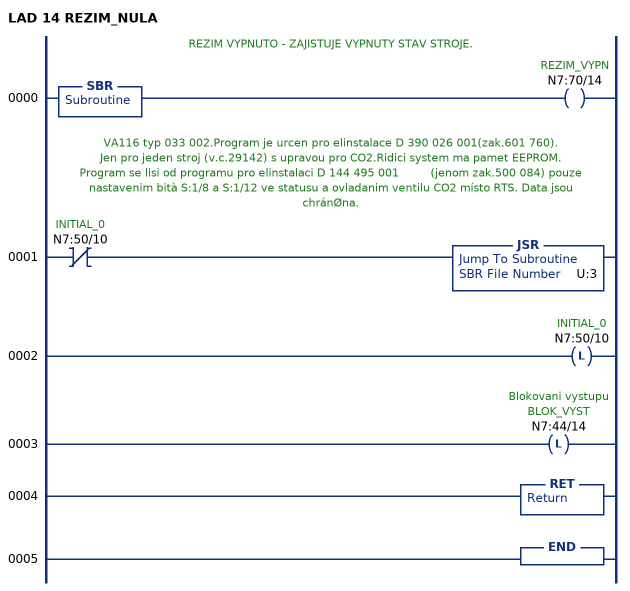
% Rung: 0 %
% REZIM VYPNUTO - ZAJISTUJE VYPNUTY STAV STROJE. %
SOR SBR OTE N7:70/14 EOR
%   N7:70/14  REZIM_VYPN %
% Rung: 1 %
% VA116 typ 033 002.Program je urcen pro elinstalace D 390 026 001(zak.601 760).
% Jen pro jeden stroj (v.c.29142) s upravou pro CO2.Ridici system ma pamet EEPROM. Program se lisi od programu pro elinstalaci D 144 495 001         (jenom zak.500 084) pouze nastavenim bità S:1/8 a S:1/12 ve statusu a ovladanim ventilu CO2 místo RTS. Data jsou chránØna. %
SOR XIO N7:50/10 JSR U:3 EOR
%   N7:50/10  INITIAL_0 %
%   JSR U:3  "Iniciali- zace po zapnuti ridiciho systemu" %
% Rung: 2 %
SOR OTL N7:50/10 EOR
%   N7:50/10  INITIAL_0 %
% Rung: 3 %
SOR OTL N7:44/14 EOR
%   N7:44/14  BLOK_VYST  "Blokovani vystupu" %
% Rung: 4 %
SOR RET EOR
% Rung: 5 %
SOR END EOR

LADDER 15 "STARTSTOP"
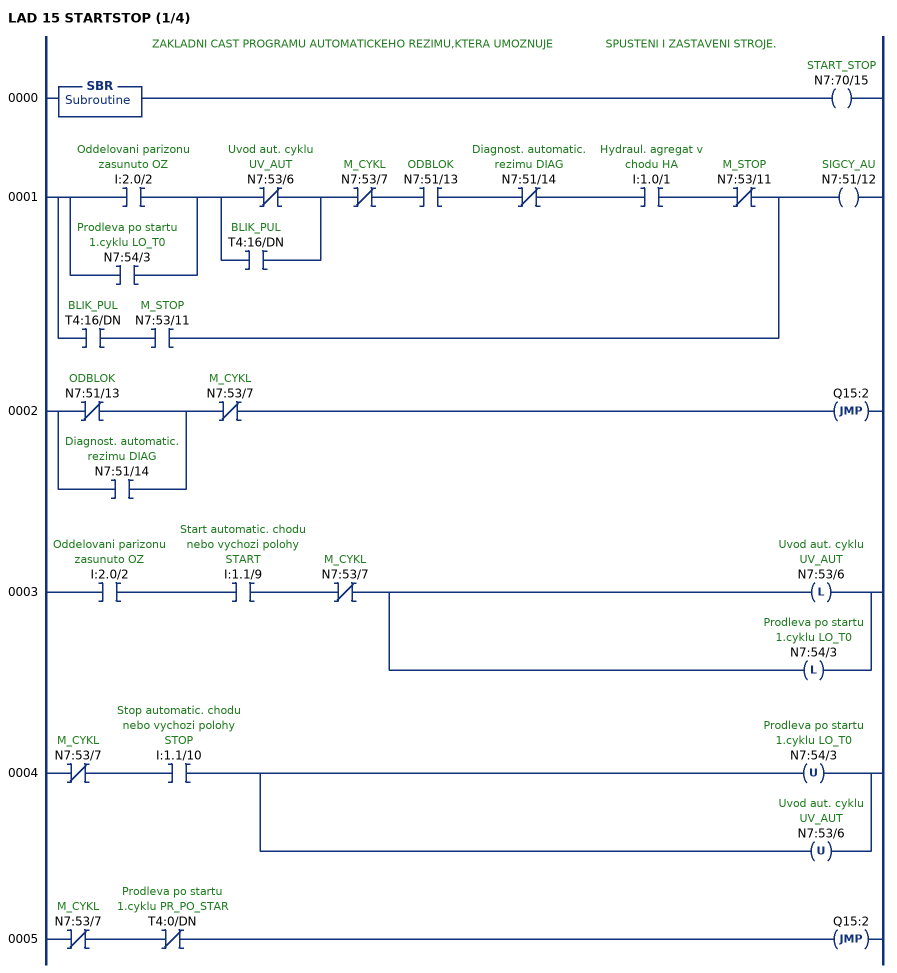
% Rung: 0 %
% ZAKLADNI CAST PROGRAMU AUTOMATICKEHO REZIMU,KTERA UMOZNUJE               SPUSTENI I ZASTAVENI STROJE. %
SOR SBR OTE N7:70/15 EOR
%   N7:70/15  START_STOP %
% Rung: 1 %
SOR BST BST XIC I:2.0/2 NXB XIC N7:54/3 BND BST XIO N7:53/6 NXB XIC T4:16/DN BND XIO N7:53/7 XIC N7:51/13 XIO N7:51/14 XIC I:1.0/1 XIO N7:53/11 NXB XIC T4:16/DN XIC N7:53/11 BND OTE N7:51/12 EOR
%   I:2.0/2  OZ  "Oddelovani parizonu zasunuto" %
%   N7:54/3  LO_T0  "Prodleva po startu 1.cyklu" %
%   N7:53/6  UV_AUT  "Uvod aut. cyklu" %
%   T4:16/DN  BLIK_PUL %
%   N7:53/7  M_CYKL %
%   N7:51/13  ODBLOK %
%   N7:51/14  DIAG  "Diagnost. automatic. rezimu" %
%   I:1.0/1  HA  "Hydraul. agregat v chodu" %
%   N7:53/11  M_STOP %
%   N7:51/12  SIGCY_AU %
% Rung: 2 %
SOR BST XIO N7:51/13 NXB XIC N7:51/14 BND XIO N7:53/7 JMP Q15:2 EOR
%   N7:51/13  ODBLOK %
%   N7:51/14  DIAG  "Diagnost. automatic. rezimu" %
%   N7:53/7  M_CYKL %
% Rung: 3 %
SOR XIC I:2.0/2 XIC I:1.1/9 XIO N7:53/7 BST OTL N7:53/6 NXB OTL N7:54/3 BND EOR
%   I:2.0/2  OZ  "Oddelovani parizonu zasunuto" %
%   I:1.1/9  START  "Start automatic. chodu nebo vychozi polohy" %
%   N7:53/7  M_CYKL %
%   N7:53/6  UV_AUT  "Uvod aut. cyklu" %
%   N7:54/3  LO_T0  "Prodleva po startu 1.cyklu" %
% Rung: 4 %
SOR XIO N7:53/7 XIC I:1.1/10 BST OTU N7:54/3 NXB OTU N7:53/6 BND EOR
%   N7:53/7  M_CYKL %
%   I:1.1/10  STOP  "Stop automatic. chodu nebo vychozi polohy" %
%   N7:54/3  LO_T0  "Prodleva po startu 1.cyklu" %
%   N7:53/6  UV_AUT  "Uvod aut. cyklu" %
% Rung: 5 %
SOR XIO N7:53/7 XIO T4:0/DN JMP Q15:2 EOR
%   N7:53/7  M_CYKL %
%   T4:0/DN  PR_PO_STAR  "Prodleva po startu 1.cyklu" %

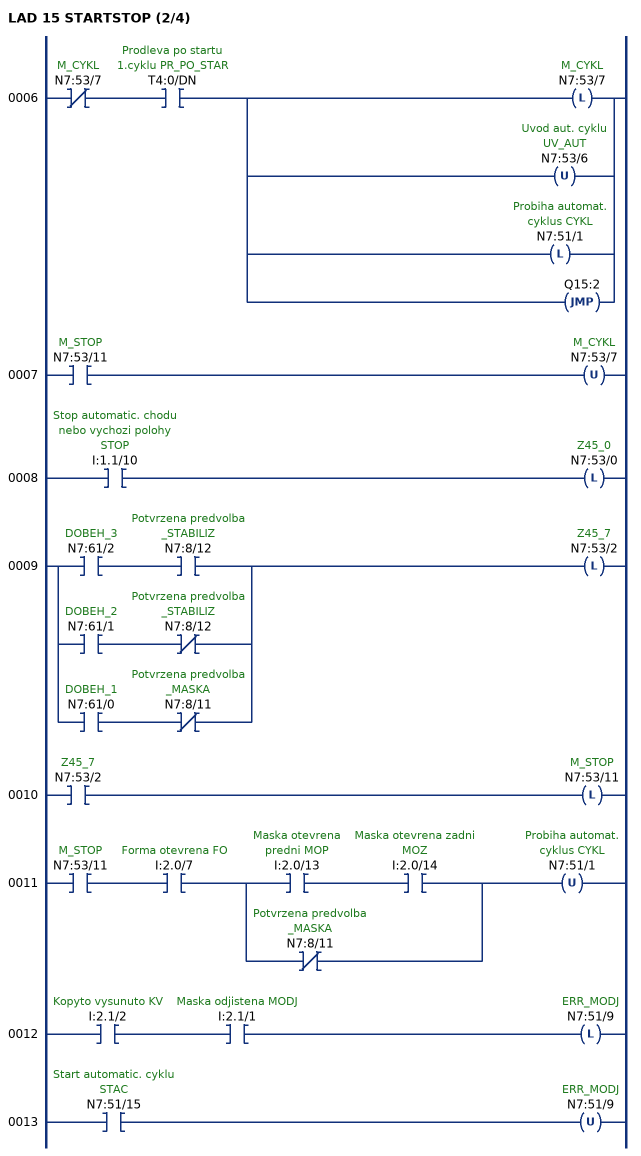
% Rung: 6 %
SOR XIO N7:53/7 XIC T4:0/DN BST OTL N7:53/7 NXB OTU N7:53/6 NXB OTL N7:51/1 NXB JMP Q15:2 BND EOR
%   N7:53/7  M_CYKL %
%   T4:0/DN  PR_PO_STAR  "Prodleva po startu 1.cyklu" %
%   N7:53/6  UV_AUT  "Uvod aut. cyklu" %
%   N7:51/1  CYKL  "Probiha automat. cyklus" %
% Rung: 7 %
SOR XIC N7:53/11 OTU N7:53/7 EOR
%   N7:53/11  M_STOP %
%   N7:53/7  M_CYKL %
% Rung: 8 %
SOR XIC I:1.1/10 OTL N7:53/0 EOR
%   I:1.1/10  STOP  "Stop automatic. chodu nebo vychozi polohy" %
%   N7:53/0  Z45_0 %
% Rung: 9 %
SOR BST XIC N7:61/2 XIC N7:8/12 NXB XIC N7:61/1 XIO N7:8/12 NXB XIC N7:61/0 XIO N7:8/11 BND OTL N7:53/2 EOR
%   N7:61/2  DOBEH_3 %
%   N7:8/12  _STABILIZ  "Potvrzena predvolba" %
%   N7:61/1  DOBEH_2 %
%   N7:61/0  DOBEH_1 %
%   N7:8/11  _MASKA  "Potvrzena predvolba" %
%   N7:53/2  Z45_7 %
% Rung: 10 %
SOR XIC N7:53/2 OTL N7:53/11 EOR
%   N7:53/2  Z45_7 %
%   N7:53/11  M_STOP %
% Rung: 11 %
SOR XIC N7:53/11 XIC I:2.0/7 BST XIC I:2.0/13 XIC I:2.0/14 NXB XIO N7:8/11 BND OTU N7:51/1 EOR
%   N7:53/11  M_STOP %
%   I:2.0/7  FO  "Forma otevrena" %
%   I:2.0/13  MOP  "Maska otevrena predni" %
%   I:2.0/14  MOZ  "Maska otevrena zadni" %
%   N7:8/11  _MASKA  "Potvrzena predvolba" %
%   N7:51/1  CYKL  "Probiha automat. cyklus" %
% Rung: 12 %
SOR XIC I:2.1/2 XIC I:2.1/1 OTL N7:51/9 EOR
%   I:2.1/2  KV  "Kopyto vysunuto" %
%   I:2.1/1  MODJ  "Maska odjistena" %
%   N7:51/9  ERR_MODJ %
% Rung: 13 %
SOR XIC N7:51/15 OTU N7:51/9 EOR
%   N7:51/15  STAC  "Start automatic. cyklu" %
%   N7:51/9  ERR_MODJ %

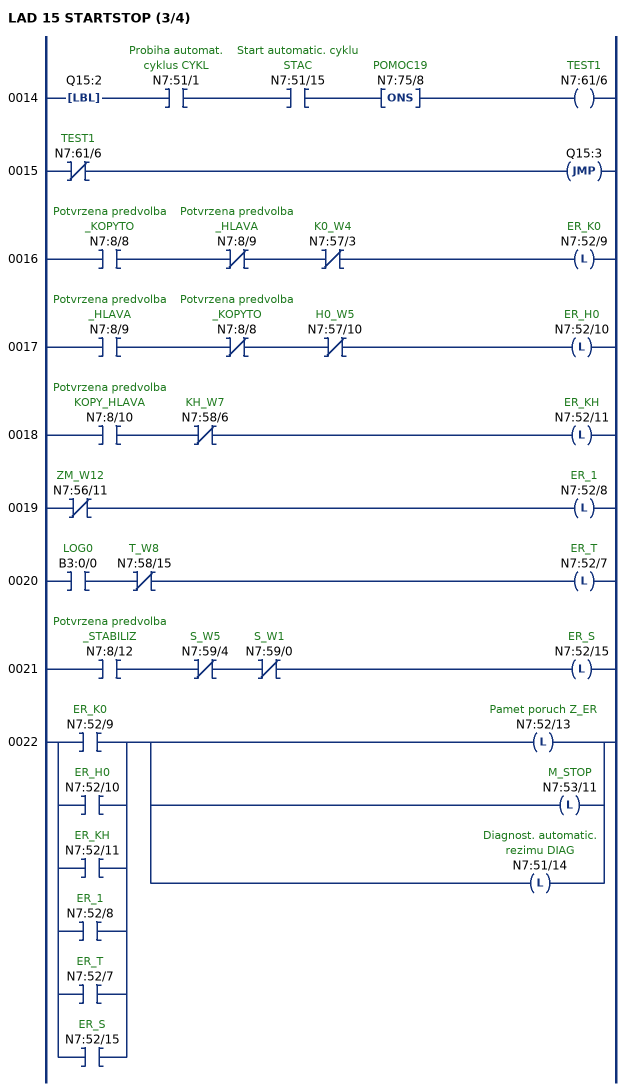
% Rung: 14 %
SOR LBL Q15:2 XIC N7:51/1 XIC N7:51/15 OSR N7:75/8 OTE N7:61/6 EOR
%   N7:51/1  CYKL  "Probiha automat. cyklus" %
%   N7:51/15  STAC  "Start automatic. cyklu" %
%   N7:75/8  POMOC19 %
%   N7:61/6  TEST1 %
% Rung: 15 %
SOR XIO N7:61/6 JMP Q15:3 EOR
%   N7:61/6  TEST1 %
% Rung: 16 %
SOR XIC N7:8/8 XIO N7:8/9 XIO N7:57/3 OTL N7:52/9 EOR
%   N7:8/8  _KOPYTO  "Potvrzena predvolba" %
%   N7:8/9  _HLAVA  "Potvrzena predvolba" %
%   N7:57/3  K0_W4 %
%   N7:52/9  ER_K0 %
% Rung: 17 %
SOR XIC N7:8/9 XIO N7:8/8 XIO N7:57/10 OTL N7:52/10 EOR
%   N7:8/9  _HLAVA  "Potvrzena predvolba" %
%   N7:8/8  _KOPYTO  "Potvrzena predvolba" %
%   N7:57/10  H0_W5 %
%   N7:52/10  ER_H0 %
% Rung: 18 %
SOR XIC N7:8/10 XIO N7:58/6 OTL N7:52/11 EOR
%   N7:8/10  KOPY_HLAVA  "Potvrzena predvolba" %
%   N7:58/6  KH_W7 %
%   N7:52/11  ER_KH %
% Rung: 19 %
SOR XIO N7:56/11 OTL N7:52/8 EOR
%   N7:56/11  ZM_W12 %
%   N7:52/8  ER_1 %
% Rung: 20 %
SOR XIC B3:0/0 XIO N7:58/15 OTL N7:52/7 EOR
%   B3:0/0  LOG0 %
%   N7:58/15  T_W8 %
%   N7:52/7  ER_T %
% Rung: 21 %
SOR XIC N7:8/12 XIO N7:59/4 XIO N7:59/0 OTL N7:52/15 EOR
%   N7:8/12  _STABILIZ  "Potvrzena predvolba" %
%   N7:59/4  S_W5 %
%   N7:59/0  S_W1 %
%   N7:52/15  ER_S %
% Rung: 22 %
SOR BST XIC N7:52/9 NXB XIC N7:52/10 NXB XIC N7:52/11 NXB XIC N7:52/8 NXB XIC N7:52/7 NXB XIC N7:52/15 BND BST OTL N7:52/13 NXB OTL N7:53/11 NXB OTL N7:51/14 BND EOR
%   N7:52/9  ER_K0 %
%   N7:52/10  ER_H0 %
%   N7:52/11  ER_KH %
%   N7:52/8  ER_1 %
%   N7:52/7  ER_T %
%   N7:52/15  ER_S %
%   N7:52/13  Z_ER  "Pamet poruch" %
%   N7:53/11  M_STOP %
%   N7:51/14  DIAG  "Diagnost. automatic. rezimu" %

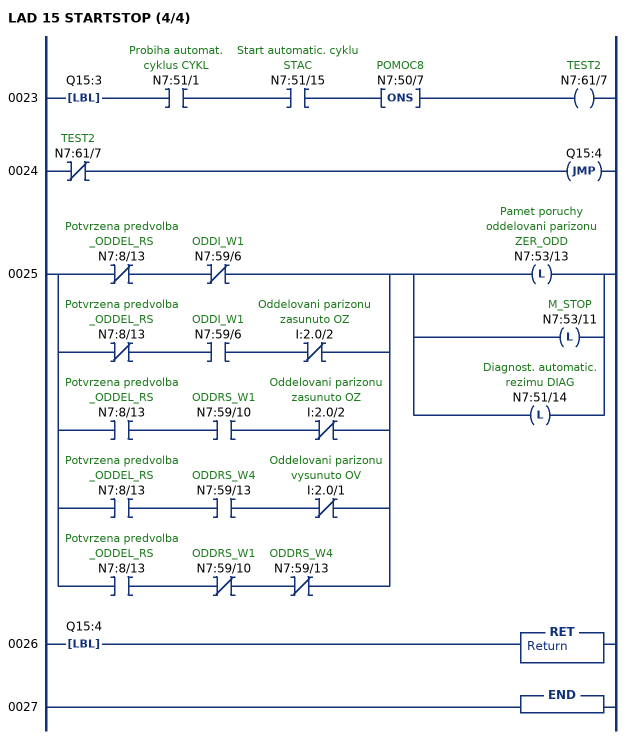
% Rung: 23 %
SOR LBL Q15:3 XIC N7:51/1 XIC N7:51/15 OSR N7:50/7 OTE N7:61/7 EOR
%   N7:51/1  CYKL  "Probiha automat. cyklus" %
%   N7:51/15  STAC  "Start automatic. cyklu" %
%   N7:50/7  POMOC8 %
%   N7:61/7  TEST2 %
% Rung: 24 %
SOR XIO N7:61/7 JMP Q15:4 EOR
%   N7:61/7  TEST2 %
% Rung: 25 %
SOR BST XIO N7:8/13 XIO N7:59/6 NXB XIO N7:8/13 XIC N7:59/6 XIO I:2.0/2 NXB XIC N7:8/13 XIC N7:59/10 XIO I:2.0/2 NXB XIC N7:8/13 XIC N7:59/13 XIO I:2.0/1 NXB XIC N7:8/13 XIO N7:59/10 XIO N7:59/13 BND BST OTL N7:53/13 NXB OTL N7:53/11 NXB OTL N7:51/14 BND EOR
%   N7:8/13  _ODDEL_RS  "Potvrzena predvolba" %
%   N7:59/6  ODDI_W1 %
%   I:2.0/2  OZ  "Oddelovani parizonu zasunuto" %
%   N7:59/10  ODDRS_W1 %
%   N7:59/13  ODDRS_W4 %
%   I:2.0/1  OV  "Oddelovani parizonu vysunuto" %
%   N7:53/13  ZER_ODD  "Pamet poruchy oddelovani parizonu" %
%   N7:53/11  M_STOP %
%   N7:51/14  DIAG  "Diagnost. automatic. rezimu" %
% Rung: 26 %
SOR LBL Q15:4 RET EOR
% Rung: 27 %
SOR END EOR

LADDER 16 "ZAKL_MECH"
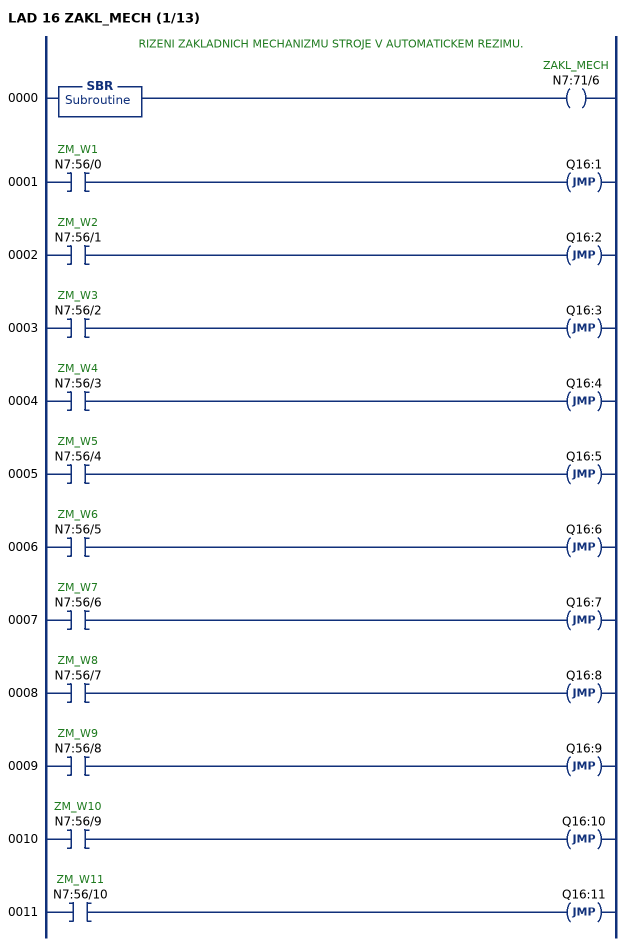
% Rung: 0 %
% RIZENI ZAKLADNICH MECHANIZMU STROJE V AUTOMATICKEM REZIMU. %
SOR SBR OTE N7:71/6 EOR
%   N7:71/6  ZAKL_MECH %
% Rung: 1 %
SOR XIC N7:56/0 JMP Q16:1 EOR
%   N7:56/0  ZM_W1 %
% Rung: 2 %
SOR XIC N7:56/1 JMP Q16:2 EOR
%   N7:56/1  ZM_W2 %
% Rung: 3 %
SOR XIC N7:56/2 JMP Q16:3 EOR
%   N7:56/2  ZM_W3 %
% Rung: 4 %
SOR XIC N7:56/3 JMP Q16:4 EOR
%   N7:56/3  ZM_W4 %
% Rung: 5 %
SOR XIC N7:56/4 JMP Q16:5 EOR
%   N7:56/4  ZM_W5 %
% Rung: 6 %
SOR XIC N7:56/5 JMP Q16:6 EOR
%   N7:56/5  ZM_W6 %
% Rung: 7 %
SOR XIC N7:56/6 JMP Q16:7 EOR
%   N7:56/6  ZM_W7 %
% Rung: 8 %
SOR XIC N7:56/7 JMP Q16:8 EOR
%   N7:56/7  ZM_W8 %
% Rung: 9 %
SOR XIC N7:56/8 JMP Q16:9 EOR
%   N7:56/8  ZM_W9 %
% Rung: 10 %
SOR XIC N7:56/9 JMP Q16:10 EOR
%   N7:56/9  ZM_W10 %
% Rung: 11 %
SOR XIC N7:56/10 JMP Q16:11 EOR
%   N7:56/10  ZM_W11 %

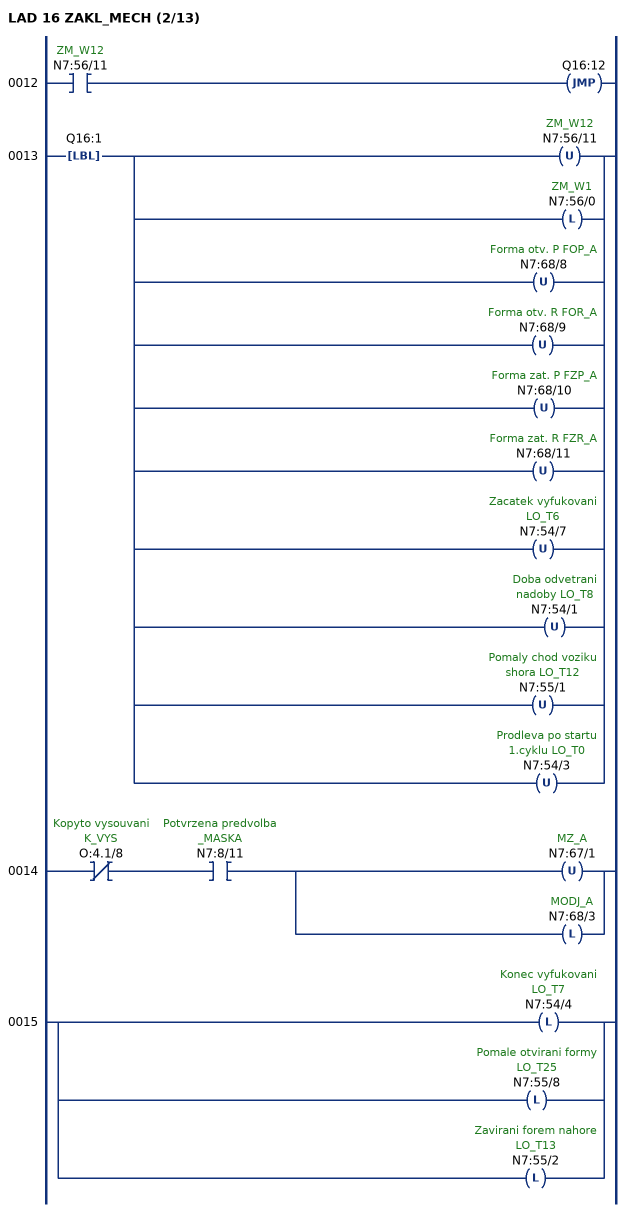
% Rung: 12 %
SOR XIC N7:56/11 JMP Q16:12 EOR
%   N7:56/11  ZM_W12 %
% Rung: 13 %
SOR LBL Q16:1 BST BST OTU N7:56/11 NXB OTL N7:56/0 BND NXB OTU N7:68/8 NXB OTU N7:68/9 NXB OTU N7:68/10 NXB OTU N7:68/11 NXB OTU N7:54/7 NXB OTU N7:54/1 NXB OTU N7:55/1 NXB OTU N7:54/3 BND EOR
%   N7:56/11  ZM_W12 %
%   N7:56/0  ZM_W1 %
%   N7:68/8  FOP_A  "Forma otv. P" %
%   N7:68/9  FOR_A  "Forma otv. R" %
%   N7:68/10  FZP_A  "Forma zat. P" %
%   N7:68/11  FZR_A  "Forma zat. R" %
%   N7:54/7  LO_T6  "Zacatek vyfukovani" %
%   N7:54/1  LO_T8  "Doba odvetrani nadoby" %
%   N7:55/1  LO_T12  "Pomaly chod voziku shora" %
%   N7:54/3  LO_T0  "Prodleva po startu 1.cyklu" %
% Rung: 14 %
SOR XIO O:4.1/8 XIC N7:8/11 BST OTU N7:67/1 NXB OTL N7:68/3 BND EOR
%   O:4.1/8  K_VYS  "Kopyto vysouvani" %
%   N7:8/11  _MASKA  "Potvrzena predvolba" %
%   N7:67/1  MZ_A %
%   N7:68/3  MODJ_A %
% Rung: 15 %
SOR BST OTL N7:54/4 NXB OTL N7:55/8 NXB OTL N7:55/2 BND EOR
%   N7:54/4  LO_T7  "Konec vyfukovani" %
%   N7:55/8  LO_T25  "Pomale otvirani formy" %
%   N7:55/2  LO_T13  "Zavirani forem nahore" %

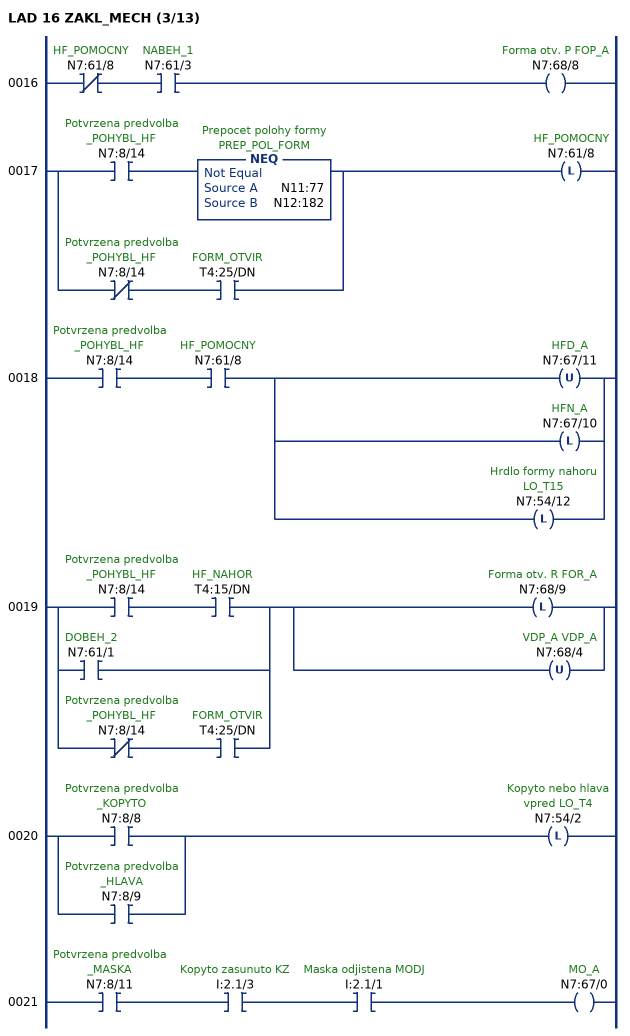
% Rung: 16 %
SOR XIO N7:61/8 XIC N7:61/3 OTE N7:68/8 EOR
%   N7:61/8  HF_POMOCNY %
%   N7:61/3  NABEH_1 %
%   N7:68/8  FOP_A  "Forma otv. P" %
% Rung: 17 %
SOR BST XIC N7:8/14 NEQ N11:77 N12:182 NXB XIO N7:8/14 XIC T4:25/DN BND OTL N7:61/8 EOR
%   N7:8/14  _POHYBL_HF  "Potvrzena predvolba" %
%   N11:77  PREP_POL_FORM  "Prepocet polohy formy" %
%   T4:25/DN  FORM_OTVIR %
%   N7:61/8  HF_POMOCNY %
% Rung: 18 %
SOR XIC N7:8/14 XIC N7:61/8 BST OTU N7:67/11 NXB OTL N7:67/10 NXB OTL N7:54/12 BND EOR
%   N7:8/14  _POHYBL_HF  "Potvrzena predvolba" %
%   N7:61/8  HF_POMOCNY %
%   N7:67/11  HFD_A %
%   N7:67/10  HFN_A %
%   N7:54/12  LO_T15  "Hrdlo formy nahoru" %
% Rung: 19 %
SOR BST XIC N7:8/14 XIC T4:15/DN NXB XIC N7:61/1 NXB XIO N7:8/14 XIC T4:25/DN BND BST OTL N7:68/9 NXB OTU N7:68/4 BND EOR
%   N7:8/14  _POHYBL_HF  "Potvrzena predvolba" %
%   T4:15/DN  HF_NAHOR %
%   N7:61/1  DOBEH_2 %
%   T4:25/DN  FORM_OTVIR %
%   N7:68/9  FOR_A  "Forma otv. R" %
%   N7:68/4  VDP_A  "VDP_A" %
% Rung: 20 %
SOR BST XIC N7:8/8 NXB XIC N7:8/9 BND OTL N7:54/2 EOR
%   N7:8/8  _KOPYTO  "Potvrzena predvolba" %
%   N7:8/9  _HLAVA  "Potvrzena predvolba" %
%   N7:54/2  LO_T4  "Kopyto nebo hlava vpred" %
% Rung: 21 %
SOR XIC N7:8/11 XIC I:2.1/3 XIC I:2.1/1 OTE N7:67/0 EOR
%   N7:8/11  _MASKA  "Potvrzena predvolba" %
%   I:2.1/3  KZ  "Kopyto zasunuto" %
%   I:2.1/1  MODJ  "Maska odjistena" %
%   N7:67/0  MO_A %

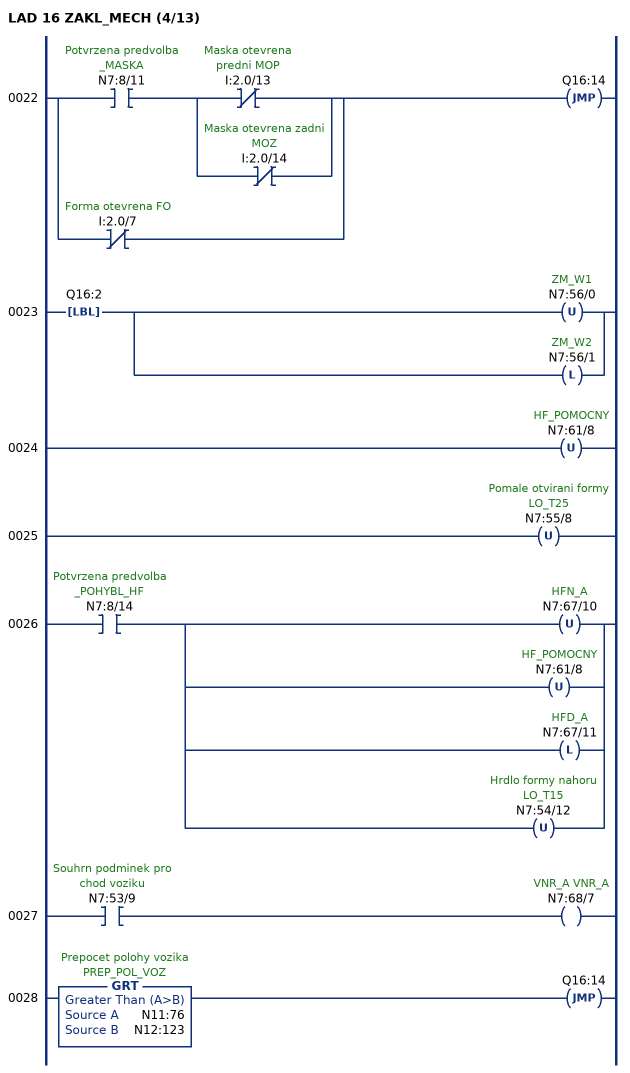
% Rung: 22 %
SOR BST XIC N7:8/11 BST XIO I:2.0/13 NXB XIO I:2.0/14 BND NXB XIO I:2.0/7 BND JMP Q16:14 EOR
%   N7:8/11  _MASKA  "Potvrzena predvolba" %
%   I:2.0/13  MOP  "Maska otevrena predni" %
%   I:2.0/14  MOZ  "Maska otevrena zadni" %
%   I:2.0/7  FO  "Forma otevrena" %
% Rung: 23 %
SOR LBL Q16:2 BST OTU N7:56/0 NXB OTL N7:56/1 BND EOR
%   N7:56/0  ZM_W1 %
%   N7:56/1  ZM_W2 %
% Rung: 24 %
SOR OTU N7:61/8 EOR
%   N7:61/8  HF_POMOCNY %
% Rung: 25 %
SOR OTU N7:55/8 EOR
%   N7:55/8  LO_T25  "Pomale otvirani formy" %
% Rung: 26 %
SOR XIC N7:8/14 BST OTU N7:67/10 NXB OTU N7:61/8 NXB OTL N7:67/11 NXB OTU N7:54/12 BND EOR
%   N7:8/14  _POHYBL_HF  "Potvrzena predvolba" %
%   N7:67/10  HFN_A %
%   N7:61/8  HF_POMOCNY %
%   N7:67/11  HFD_A %
%   N7:54/12  LO_T15  "Hrdlo formy nahoru" %
% Rung: 27 %
SOR XIC N7:53/9 OTE N7:68/7 EOR
%   N7:53/9  "Souhrn podminek pro chod voziku" %
%   N7:68/7  VNR_A  "VNR_A" %
% Rung: 28 %
SOR GRT N11:76 N12:123 JMP Q16:14 EOR
%   N11:76  PREP_POL_VOZ  "Prepocet polohy vozika" %
%   N12:123  N123  "Žiadana poloha vozika c.4 hore" %

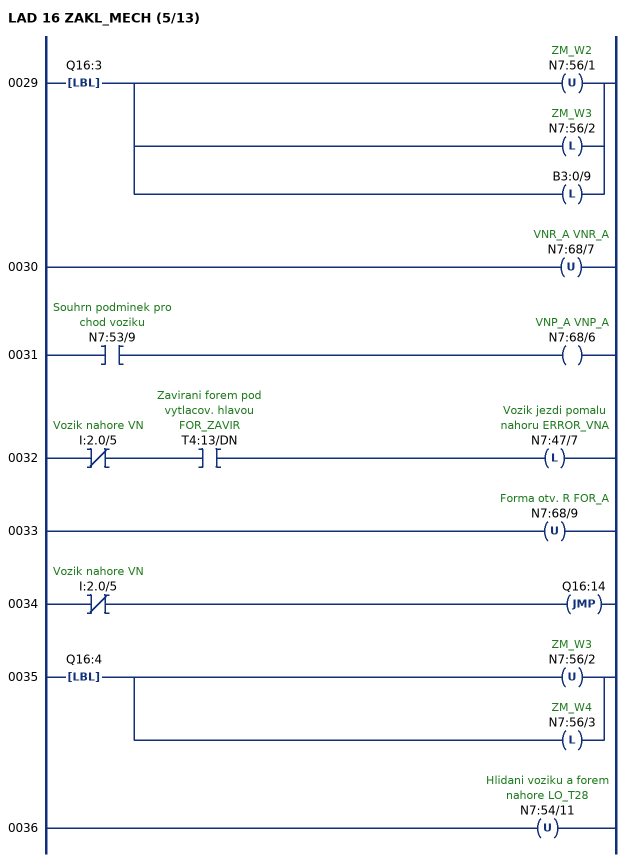
% Rung: 29 %
SOR LBL Q16:3 BST OTU N7:56/1 NXB OTL N7:56/2 NXB OTL B3:0/9 BND EOR
%   N7:56/1  ZM_W2 %
%   N7:56/2  ZM_W3 %
% Rung: 30 %
SOR OTU N7:68/7 EOR
%   N7:68/7  VNR_A  "VNR_A" %
% Rung: 31 %
SOR XIC N7:53/9 OTE N7:68/6 EOR
%   N7:53/9  "Souhrn podminek pro chod voziku" %
%   N7:68/6  VNP_A  "VNP_A" %
% Rung: 32 %
SOR XIO I:2.0/5 XIC T4:13/DN OTL N7:47/7 EOR
%   I:2.0/5  VN  "Vozik nahore" %
%   T4:13/DN  FOR_ZAVIR  "Zavirani forem pod vytlacov. hlavou" %
%   N7:47/7  ERROR_VNA  "Vozik jezdi pomalu nahoru" %
% Rung: 33 %
SOR OTU N7:68/9 EOR
%   N7:68/9  FOR_A  "Forma otv. R" %
% Rung: 34 %
SOR XIO I:2.0/5 JMP Q16:14 EOR
%   I:2.0/5  VN  "Vozik nahore" %
% Rung: 35 %
SOR LBL Q16:4 BST OTU N7:56/2 NXB OTL N7:56/3 BND EOR
%   N7:56/2  ZM_W3 %
%   N7:56/3  ZM_W4 %
% Rung: 36 %
SOR OTU N7:54/11 EOR
%   N7:54/11  LO_T28  "Hlidani voziku a forem nahore" %

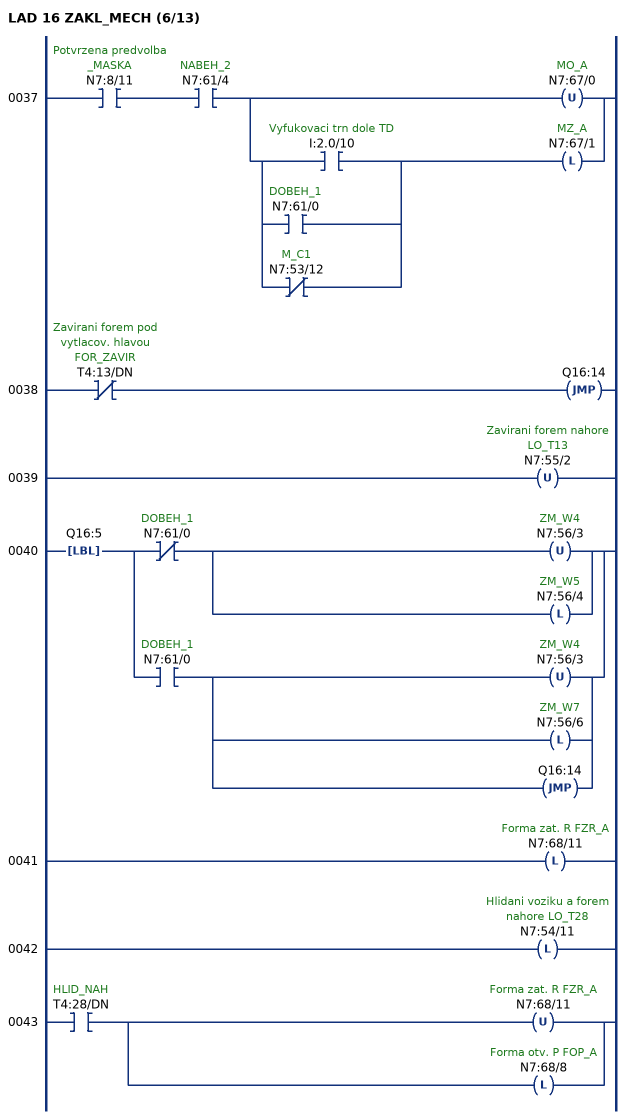
% Rung: 37 %
SOR XIC N7:8/11 XIC N7:61/4 BST OTU N7:67/0 NXB BST XIC I:2.0/10 NXB XIC N7:61/0 NXB XIO N7:53/12 BND OTL N7:67/1 BND EOR
%   N7:8/11  _MASKA  "Potvrzena predvolba" %
%   N7:61/4  NABEH_2 %
%   N7:67/0  MO_A %
%   I:2.0/10  TD  "Vyfukovaci trn dole" %
%   N7:61/0  DOBEH_1 %
%   N7:53/12  M_C1 %
%   N7:67/1  MZ_A %
% Rung: 38 %
SOR XIO T4:13/DN JMP Q16:14 EOR
%   T4:13/DN  FOR_ZAVIR  "Zavirani forem pod vytlacov. hlavou" %
% Rung: 39 %
SOR OTU N7:55/2 EOR
%   N7:55/2  LO_T13  "Zavirani forem nahore" %
% Rung: 40 %
SOR LBL Q16:5 BST XIO N7:61/0 BST OTU N7:56/3 NXB OTL N7:56/4 BND NXB XIC N7:61/0 BST OTU N7:56/3 NXB OTL N7:56/6 NXB JMP Q16:14 BND BND EOR
%   N7:61/0  DOBEH_1 %
%   N7:56/3  ZM_W4 %
%   N7:56/4  ZM_W5 %
%   N7:56/6  ZM_W7 %
% Rung: 41 %
SOR OTL N7:68/11 EOR
%   N7:68/11  FZR_A  "Forma zat. R" %
% Rung: 42 %
SOR OTL N7:54/11 EOR
%   N7:54/11  LO_T28  "Hlidani voziku a forem nahore" %
% Rung: 43 %
SOR XIC T4:28/DN BST OTU N7:68/11 NXB OTL N7:68/8 BND EOR
%   T4:28/DN  HLID_NAH %
%   N7:68/11  FZR_A  "Forma zat. R" %
%   N7:68/8  FOP_A  "Forma otv. P" %

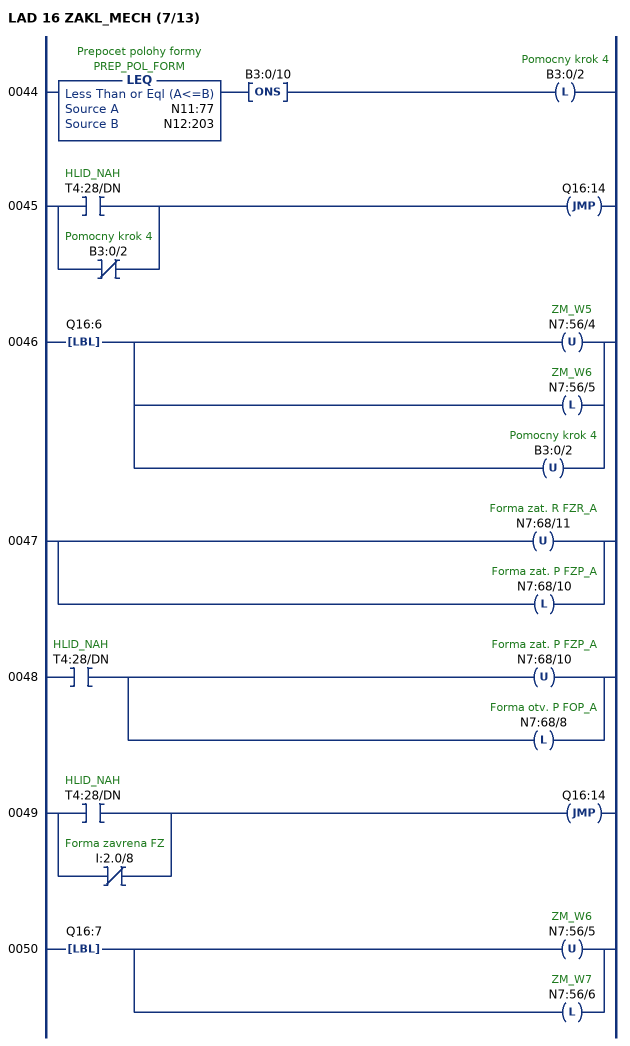
% Rung: 44 %
SOR LEQ N11:77 N12:203 OSR B3:0/10 OTL B3:0/2 EOR
%   N11:77  PREP_POL_FORM  "Prepocet polohy formy" %
%   B3:0/2  "Pomocny krok 4" %
% Rung: 45 %
SOR BST XIC T4:28/DN NXB XIO B3:0/2 BND JMP Q16:14 EOR
%   T4:28/DN  HLID_NAH %
%   B3:0/2  "Pomocny krok 4" %
% Rung: 46 %
SOR LBL Q16:6 BST OTU N7:56/4 NXB OTL N7:56/5 NXB OTU B3:0/2 BND EOR
%   N7:56/4  ZM_W5 %
%   N7:56/5  ZM_W6 %
%   B3:0/2  "Pomocny krok 4" %
% Rung: 47 %
SOR BST OTU N7:68/11 NXB OTL N7:68/10 BND EOR
%   N7:68/11  FZR_A  "Forma zat. R" %
%   N7:68/10  FZP_A  "Forma zat. P" %
% Rung: 48 %
SOR XIC T4:28/DN BST OTU N7:68/10 NXB OTL N7:68/8 BND EOR
%   T4:28/DN  HLID_NAH %
%   N7:68/10  FZP_A  "Forma zat. P" %
%   N7:68/8  FOP_A  "Forma otv. P" %
% Rung: 49 %
SOR BST XIC T4:28/DN NXB XIO I:2.0/8 BND JMP Q16:14 EOR
%   T4:28/DN  HLID_NAH %
%   I:2.0/8  FZ  "Forma zavrena" %
% Rung: 50 %
SOR LBL Q16:7 BST OTU N7:56/5 NXB OTL N7:56/6 BND EOR
%   N7:56/5  ZM_W6 %
%   N7:56/6  ZM_W7 %

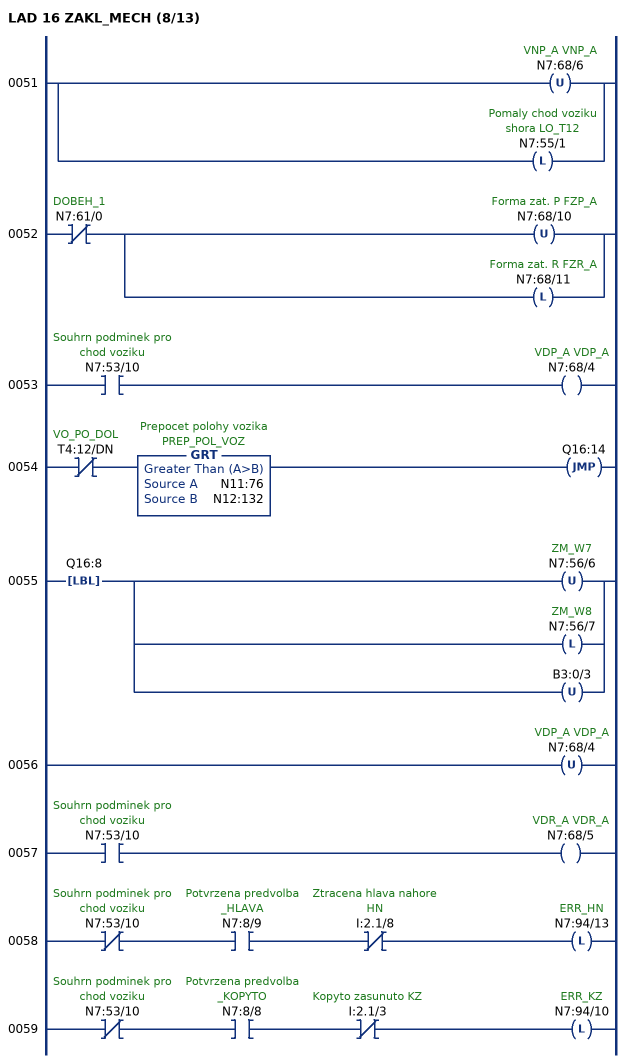
% Rung: 51 %
SOR BST OTU N7:68/6 NXB OTL N7:55/1 BND EOR
%   N7:68/6  VNP_A  "VNP_A" %
%   N7:55/1  LO_T12  "Pomaly chod voziku shora" %
% Rung: 52 %
SOR XIO N7:61/0 BST OTU N7:68/10 NXB OTL N7:68/11 BND EOR
%   N7:61/0  DOBEH_1 %
%   N7:68/10  FZP_A  "Forma zat. P" %
%   N7:68/11  FZR_A  "Forma zat. R" %
% Rung: 53 %
SOR XIC N7:53/10 OTE N7:68/4 EOR
%   N7:53/10  "Souhrn podminek pro chod voziku" %
%   N7:68/4  VDP_A  "VDP_A" %
% Rung: 54 %
SOR XIO T4:12/DN GRT N11:76 N12:132 JMP Q16:14 EOR
%   T4:12/DN  VO_PO_DOL %
%   N11:76  PREP_POL_VOZ  "Prepocet polohy vozika" %
% Rung: 55 %
SOR LBL Q16:8 BST OTU N7:56/6 NXB OTL N7:56/7 NXB OTU B3:0/3 BND EOR
%   N7:56/6  ZM_W7 %
%   N7:56/7  ZM_W8 %
% Rung: 56 %
SOR OTU N7:68/4 EOR
%   N7:68/4  VDP_A  "VDP_A" %
% Rung: 57 %
SOR XIC N7:53/10 OTE N7:68/5 EOR
%   N7:53/10  "Souhrn podminek pro chod voziku" %
%   N7:68/5  VDR_A  "VDR_A" %
% Rung: 58 %
SOR XIO N7:53/10 XIC N7:8/9 XIO I:2.1/8 OTL N7:94/13 EOR
%   N7:53/10  "Souhrn podminek pro chod voziku" %
%   N7:8/9  _HLAVA  "Potvrzena predvolba" %
%   I:2.1/8  HN  "Ztracena hlava nahore" %
%   N7:94/13  ERR_HN %
% Rung: 59 %
SOR XIO N7:53/10 XIC N7:8/8 XIO I:2.1/3 OTL N7:94/10 EOR
%   N7:53/10  "Souhrn podminek pro chod voziku" %
%   N7:8/8  _KOPYTO  "Potvrzena predvolba" %
%   I:2.1/3  KZ  "Kopyto zasunuto" %
%   N7:94/10  ERR_KZ %

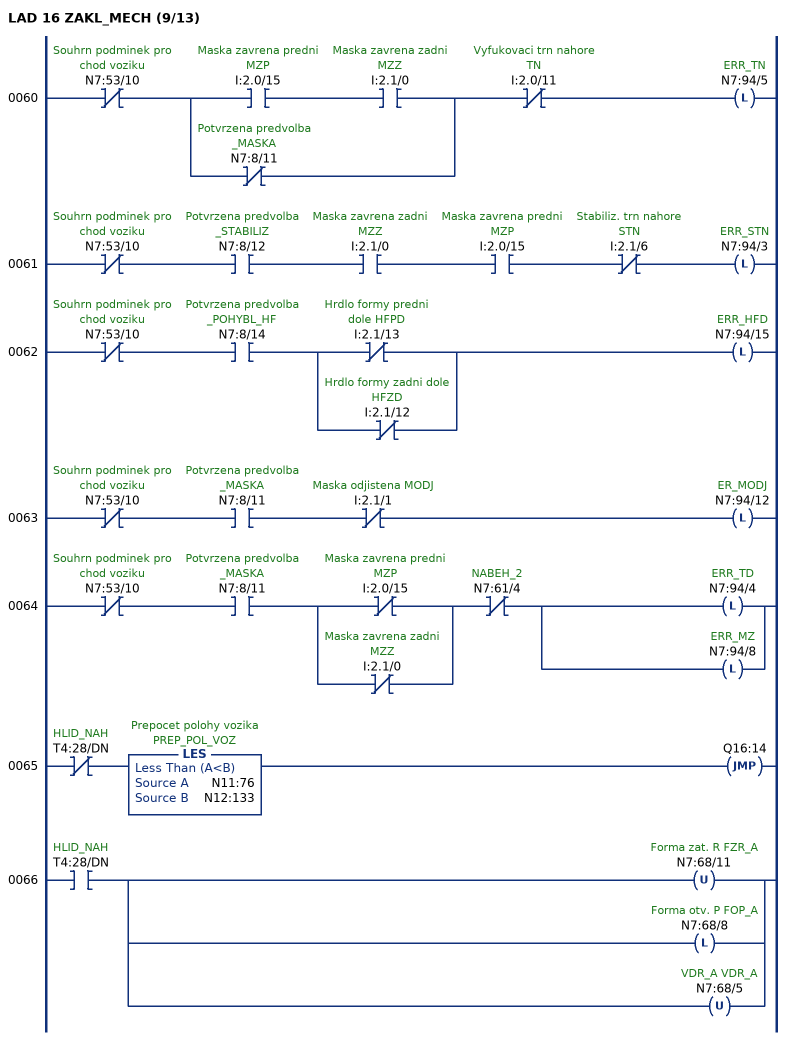
% Rung: 60 %
SOR XIO N7:53/10 BST XIC I:2.0/15 XIC I:2.1/0 NXB XIO N7:8/11 BND XIO I:2.0/11 OTL N7:94/5 EOR
%   N7:53/10  "Souhrn podminek pro chod voziku" %
%   I:2.0/15  MZP  "Maska zavrena predni" %
%   I:2.1/0  MZZ  "Maska zavrena zadni" %
%   N7:8/11  _MASKA  "Potvrzena predvolba" %
%   I:2.0/11  TN  "Vyfukovaci trn nahore" %
%   N7:94/5  ERR_TN %
% Rung: 61 %
SOR XIO N7:53/10 XIC N7:8/12 XIC I:2.1/0 XIC I:2.0/15 XIO I:2.1/6 OTL N7:94/3 EOR
%   N7:53/10  "Souhrn podminek pro chod voziku" %
%   N7:8/12  _STABILIZ  "Potvrzena predvolba" %
%   I:2.1/0  MZZ  "Maska zavrena zadni" %
%   I:2.0/15  MZP  "Maska zavrena predni" %
%   I:2.1/6  STN  "Stabiliz. trn nahore" %
%   N7:94/3  ERR_STN %
% Rung: 62 %
SOR XIO N7:53/10 XIC N7:8/14 BST XIO I:2.1/13 NXB XIO I:2.1/12 BND OTL N7:94/15 EOR
%   N7:53/10  "Souhrn podminek pro chod voziku" %
%   N7:8/14  _POHYBL_HF  "Potvrzena predvolba" %
%   I:2.1/13  HFPD  "Hrdlo formy predni dole" %
%   I:2.1/12  HFZD  "Hrdlo formy zadni dole" %
%   N7:94/15  ERR_HFD %
% Rung: 63 %
SOR XIO N7:53/10 XIC N7:8/11 XIO I:2.1/1 OTL N7:94/12 EOR
%   N7:53/10  "Souhrn podminek pro chod voziku" %
%   N7:8/11  _MASKA  "Potvrzena predvolba" %
%   I:2.1/1  MODJ  "Maska odjistena" %
%   N7:94/12  ER_MODJ %
% Rung: 64 %
SOR XIO N7:53/10 XIC N7:8/11 BST XIO I:2.0/15 NXB XIO I:2.1/0 BND XIO N7:61/4 BST OTL N7:94/4 NXB OTL N7:94/8 BND EOR
%   N7:53/10  "Souhrn podminek pro chod voziku" %
%   N7:8/11  _MASKA  "Potvrzena predvolba" %
%   I:2.0/15  MZP  "Maska zavrena predni" %
%   I:2.1/0  MZZ  "Maska zavrena zadni" %
%   N7:61/4  NABEH_2 %
%   N7:94/4  ERR_TD %
%   N7:94/8  ERR_MZ %
% Rung: 65 %
SOR XIO T4:28/DN LES N11:76 N12:133 JMP Q16:14 EOR
%   T4:28/DN  HLID_NAH %
%   N11:76  PREP_POL_VOZ  "Prepocet polohy vozika" %
% Rung: 66 %
SOR XIC T4:28/DN BST OTU N7:68/11 NXB OTL N7:68/8 NXB OTU N7:68/5 BND EOR
%   T4:28/DN  HLID_NAH %
%   N7:68/11  FZR_A  "Forma zat. R" %
%   N7:68/8  FOP_A  "Forma otv. P" %
%   N7:68/5  VDR_A  "VDR_A" %

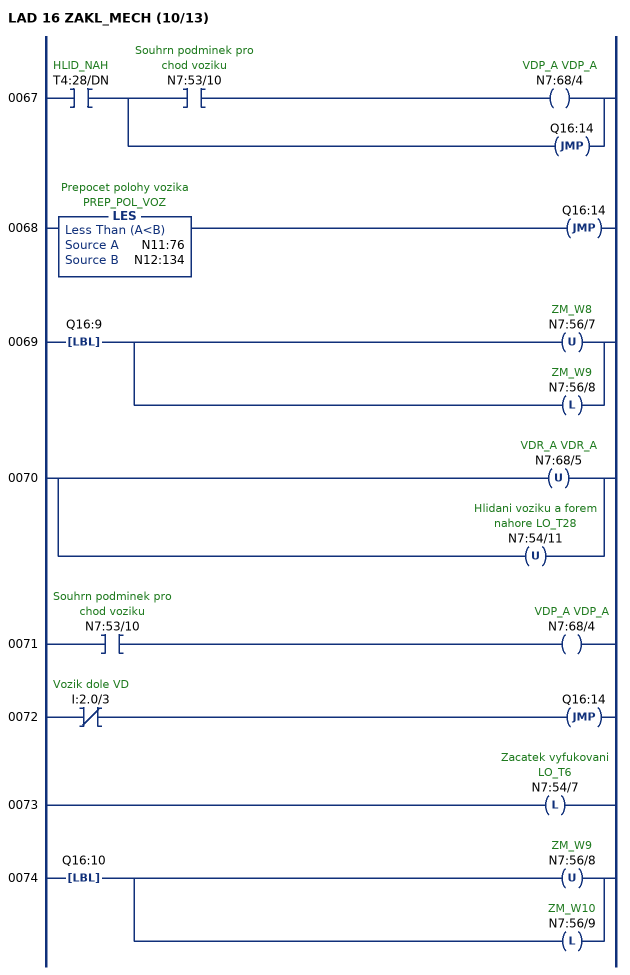
% Rung: 67 %
SOR XIC T4:28/DN BST XIC N7:53/10 OTE N7:68/4 NXB JMP Q16:14 BND EOR
%   T4:28/DN  HLID_NAH %
%   N7:53/10  "Souhrn podminek pro chod voziku" %
%   N7:68/4  VDP_A  "VDP_A" %
% Rung: 68 %
SOR LES N11:76 N12:134 JMP Q16:14 EOR
%   N11:76  PREP_POL_VOZ  "Prepocet polohy vozika" %
% Rung: 69 %
SOR LBL Q16:9 BST OTU N7:56/7 NXB OTL N7:56/8 BND EOR
%   N7:56/7  ZM_W8 %
%   N7:56/8  ZM_W9 %
% Rung: 70 %
SOR BST OTU N7:68/5 NXB OTU N7:54/11 BND EOR
%   N7:68/5  VDR_A  "VDR_A" %
%   N7:54/11  LO_T28  "Hlidani voziku a forem nahore" %
% Rung: 71 %
SOR XIC N7:53/10 OTE N7:68/4 EOR
%   N7:53/10  "Souhrn podminek pro chod voziku" %
%   N7:68/4  VDP_A  "VDP_A" %
% Rung: 72 %
SOR XIO I:2.0/3 JMP Q16:14 EOR
%   I:2.0/3  VD  "Vozik dole" %
% Rung: 73 %
SOR OTL N7:54/7 EOR
%   N7:54/7  LO_T6  "Zacatek vyfukovani" %
% Rung: 74 %
SOR LBL Q16:10 BST OTU N7:56/8 NXB OTL N7:56/9 BND EOR
%   N7:56/8  ZM_W9 %
%   N7:56/9  ZM_W10 %

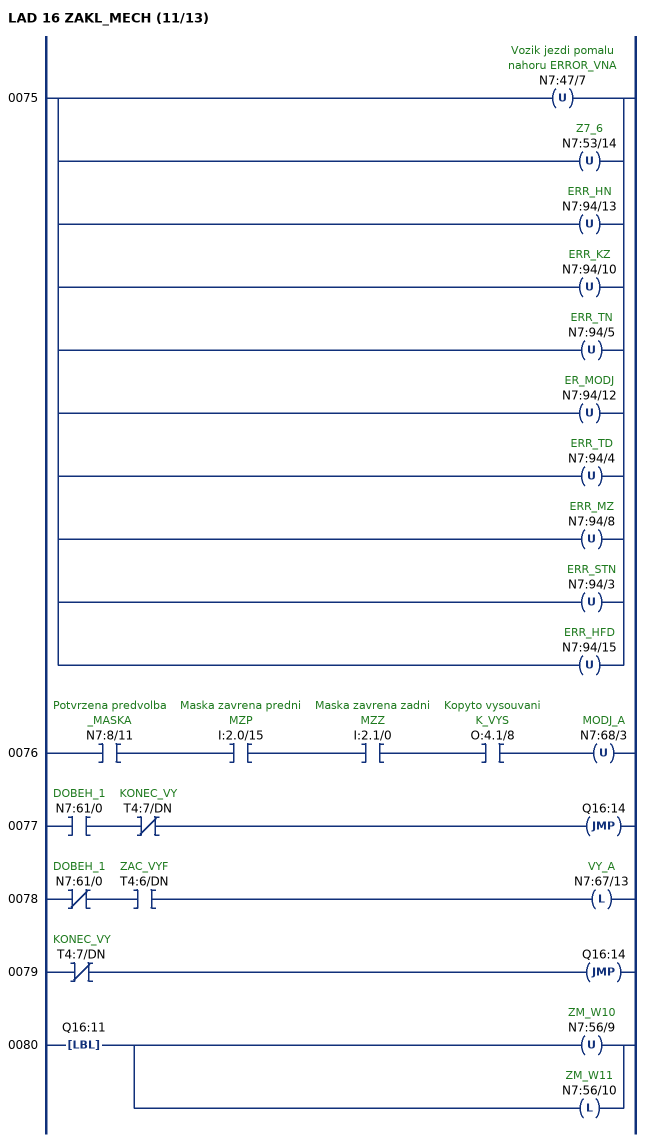
% Rung: 75 %
SOR BST OTU N7:47/7 NXB OTU N7:53/14 NXB OTU N7:94/13 NXB OTU N7:94/10 NXB OTU N7:94/5 NXB OTU N7:94/12 NXB OTU N7:94/4 NXB OTU N7:94/8 NXB OTU N7:94/3 NXB OTU N7:94/15 BND EOR
%   N7:47/7  ERROR_VNA  "Vozik jezdi pomalu nahoru" %
%   N7:53/14  Z7_6 %
%   N7:94/13  ERR_HN %
%   N7:94/10  ERR_KZ %
%   N7:94/5  ERR_TN %
%   N7:94/12  ER_MODJ %
%   N7:94/4  ERR_TD %
%   N7:94/8  ERR_MZ %
%   N7:94/3  ERR_STN %
%   N7:94/15  ERR_HFD %
% Rung: 76 %
SOR XIC N7:8/11 XIC I:2.0/15 XIC I:2.1/0 XIC O:4.1/8 OTU N7:68/3 EOR
%   N7:8/11  _MASKA  "Potvrzena predvolba" %
%   I:2.0/15  MZP  "Maska zavrena predni" %
%   I:2.1/0  MZZ  "Maska zavrena zadni" %
%   O:4.1/8  K_VYS  "Kopyto vysouvani" %
%   N7:68/3  MODJ_A %
% Rung: 77 %
SOR XIC N7:61/0 XIO T4:7/DN JMP Q16:14 EOR
%   N7:61/0  DOBEH_1 %
%   T4:7/DN  KONEC_VY %
% Rung: 78 %
SOR XIO N7:61/0 XIC T4:6/DN OTL N7:67/13 EOR
%   N7:61/0  DOBEH_1 %
%   T4:6/DN  ZAC_VYF %
%   N7:67/13  VY_A %
% Rung: 79 %
SOR XIO T4:7/DN JMP Q16:14 EOR
%   T4:7/DN  KONEC_VY %
% Rung: 80 %
SOR LBL Q16:11 BST OTU N7:56/9 NXB OTL N7:56/10 BND EOR
%   N7:56/9  ZM_W10 %
%   N7:56/10  ZM_W11 %

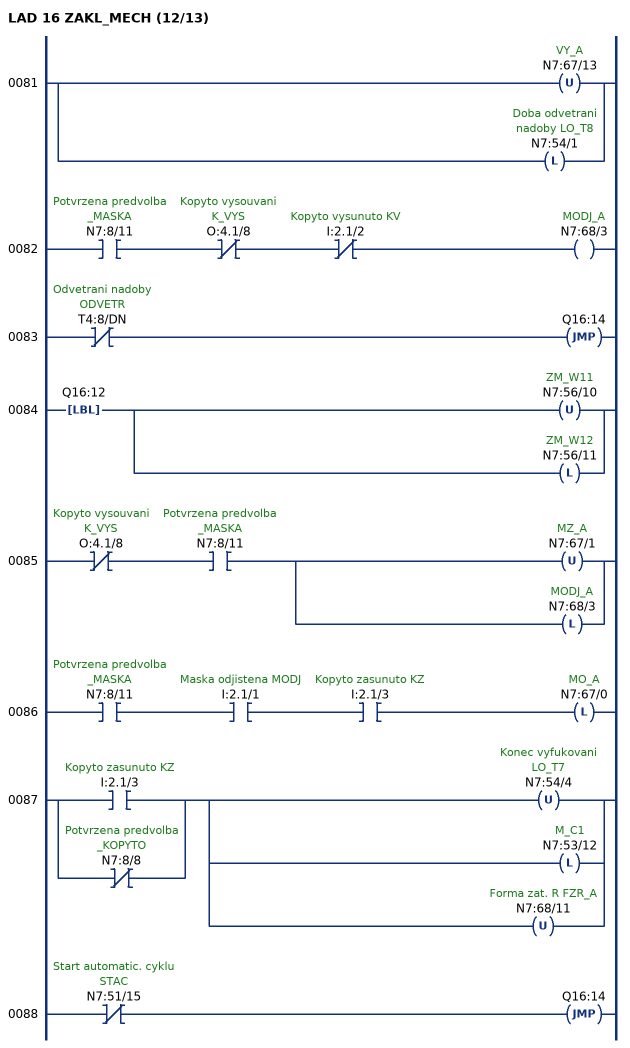
% Rung: 81 %
SOR BST OTU N7:67/13 NXB OTL N7:54/1 BND EOR
%   N7:67/13  VY_A %
%   N7:54/1  LO_T8  "Doba odvetrani nadoby" %
% Rung: 82 %
SOR XIC N7:8/11 XIO O:4.1/8 XIO I:2.1/2 OTE N7:68/3 EOR
%   N7:8/11  _MASKA  "Potvrzena predvolba" %
%   O:4.1/8  K_VYS  "Kopyto vysouvani" %
%   I:2.1/2  KV  "Kopyto vysunuto" %
%   N7:68/3  MODJ_A %
% Rung: 83 %
SOR XIO T4:8/DN JMP Q16:14 EOR
%   T4:8/DN  ODVETR  "Odvetrani nadoby" %
% Rung: 84 %
SOR LBL Q16:12 BST OTU N7:56/10 NXB OTL N7:56/11 BND EOR
%   N7:56/10  ZM_W11 %
%   N7:56/11  ZM_W12 %
% Rung: 85 %
SOR XIO O:4.1/8 XIC N7:8/11 BST OTU N7:67/1 NXB OTL N7:68/3 BND EOR
%   O:4.1/8  K_VYS  "Kopyto vysouvani" %
%   N7:8/11  _MASKA  "Potvrzena predvolba" %
%   N7:67/1  MZ_A %
%   N7:68/3  MODJ_A %
% Rung: 86 %
SOR XIC N7:8/11 XIC I:2.1/1 XIC I:2.1/3 OTL N7:67/0 EOR
%   N7:8/11  _MASKA  "Potvrzena predvolba" %
%   I:2.1/1  MODJ  "Maska odjistena" %
%   I:2.1/3  KZ  "Kopyto zasunuto" %
%   N7:67/0  MO_A %
% Rung: 87 %
SOR BST XIC I:2.1/3 NXB XIO N7:8/8 BND BST OTU N7:54/4 NXB OTL N7:53/12 NXB OTU N7:68/11 BND EOR
%   I:2.1/3  KZ  "Kopyto zasunuto" %
%   N7:8/8  _KOPYTO  "Potvrzena predvolba" %
%   N7:54/4  LO_T7  "Konec vyfukovani" %
%   N7:53/12  M_C1 %
%   N7:68/11  FZR_A  "Forma zat. R" %
% Rung: 88 %
SOR XIO N7:51/15 JMP Q16:14 EOR
%   N7:51/15  STAC  "Start automatic. cyklu" %

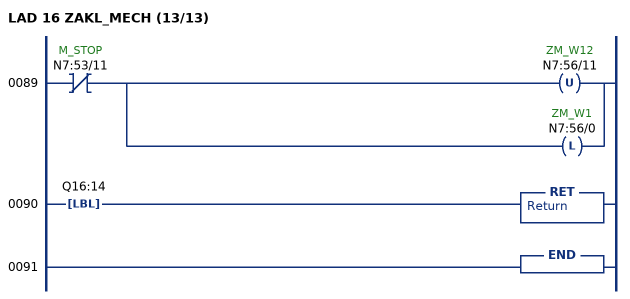
% Rung: 89 %
SOR XIO N7:53/11 BST OTU N7:56/11 NXB OTL N7:56/0 BND EOR
%   N7:53/11  M_STOP %
%   N7:56/11  ZM_W12 %
%   N7:56/0  ZM_W1 %
% Rung: 90 %
SOR LBL Q16:14 RET EOR
% Rung: 91 %
SOR END EOR

LADDER 17 "KOPYTO_SOL"
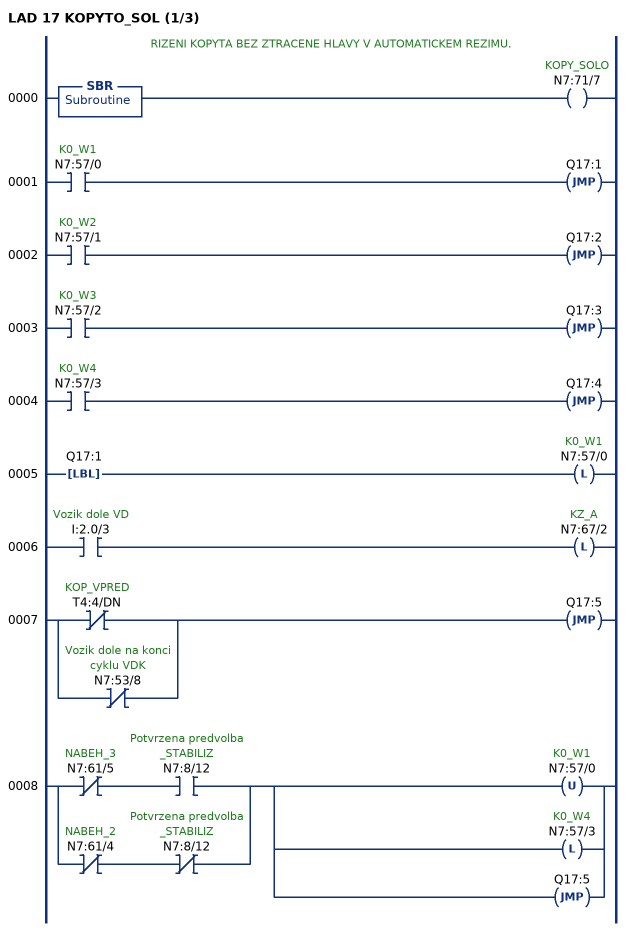
% Rung: 0 %
% RIZENI KOPYTA BEZ ZTRACENE HLAVY V AUTOMATICKEM REZIMU. %
SOR SBR OTE N7:71/7 EOR
%   N7:71/7  KOPY_SOLO %
% Rung: 1 %
SOR XIC N7:57/0 JMP Q17:1 EOR
%   N7:57/0  K0_W1 %
% Rung: 2 %
SOR XIC N7:57/1 JMP Q17:2 EOR
%   N7:57/1  K0_W2 %
% Rung: 3 %
SOR XIC N7:57/2 JMP Q17:3 EOR
%   N7:57/2  K0_W3 %
% Rung: 4 %
SOR XIC N7:57/3 JMP Q17:4 EOR
%   N7:57/3  K0_W4 %
% Rung: 5 %
SOR LBL Q17:1 OTL N7:57/0 EOR
%   N7:57/0  K0_W1 %
% Rung: 6 %
SOR XIC I:2.0/3 OTL N7:67/2 EOR
%   I:2.0/3  VD  "Vozik dole" %
%   N7:67/2  KZ_A %
% Rung: 7 %
SOR BST XIO T4:4/DN NXB XIO N7:53/8 BND JMP Q17:5 EOR
%   T4:4/DN  KOP_VPRED %
%   N7:53/8  VDK  "Vozik dole na konci cyklu" %
% Rung: 8 %
SOR BST XIO N7:61/5 XIC N7:8/12 NXB XIO N7:61/4 XIO N7:8/12 BND BST OTU N7:57/0 NXB OTL N7:57/3 NXB JMP Q17:5 BND EOR
%   N7:61/5  NABEH_3 %
%   N7:8/12  _STABILIZ  "Potvrzena predvolba" %
%   N7:61/4  NABEH_2 %
%   N7:57/0  K0_W1 %
%   N7:57/3  K0_W4 %

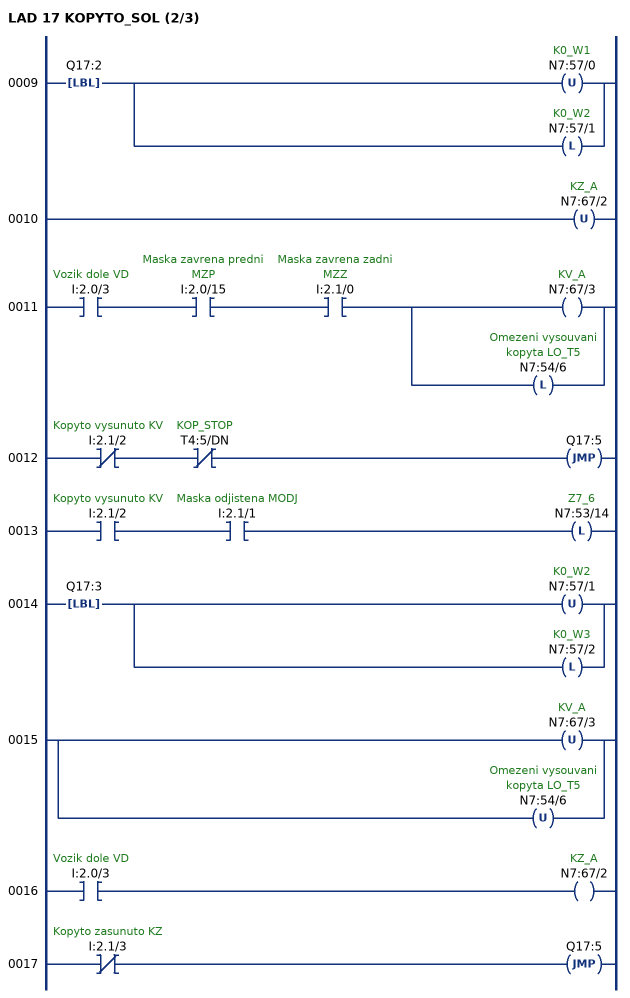
% Rung: 9 %
SOR LBL Q17:2 BST OTU N7:57/0 NXB OTL N7:57/1 BND EOR
%   N7:57/0  K0_W1 %
%   N7:57/1  K0_W2 %
% Rung: 10 %
SOR OTU N7:67/2 EOR
%   N7:67/2  KZ_A %
% Rung: 11 %
SOR XIC I:2.0/3 XIC I:2.0/15 XIC I:2.1/0 BST OTE N7:67/3 NXB OTL N7:54/6 BND EOR
%   I:2.0/3  VD  "Vozik dole" %
%   I:2.0/15  MZP  "Maska zavrena predni" %
%   I:2.1/0  MZZ  "Maska zavrena zadni" %
%   N7:67/3  KV_A %
%   N7:54/6  LO_T5  "Omezeni vysouvani kopyta" %
% Rung: 12 %
SOR XIO I:2.1/2 XIO T4:5/DN JMP Q17:5 EOR
%   I:2.1/2  KV  "Kopyto vysunuto" %
%   T4:5/DN  KOP_STOP %
% Rung: 13 %
SOR XIC I:2.1/2 XIC I:2.1/1 OTL N7:53/14 EOR
%   I:2.1/2  KV  "Kopyto vysunuto" %
%   I:2.1/1  MODJ  "Maska odjistena" %
%   N7:53/14  Z7_6 %
% Rung: 14 %
SOR LBL Q17:3 BST OTU N7:57/1 NXB OTL N7:57/2 BND EOR
%   N7:57/1  K0_W2 %
%   N7:57/2  K0_W3 %
% Rung: 15 %
SOR BST OTU N7:67/3 NXB OTU N7:54/6 BND EOR
%   N7:67/3  KV_A %
%   N7:54/6  LO_T5  "Omezeni vysouvani kopyta" %
% Rung: 16 %
SOR XIC I:2.0/3 OTE N7:67/2 EOR
%   I:2.0/3  VD  "Vozik dole" %
%   N7:67/2  KZ_A %
% Rung: 17 %
SOR XIO I:2.1/3 JMP Q17:5 EOR
%   I:2.1/3  KZ  "Kopyto zasunuto" %

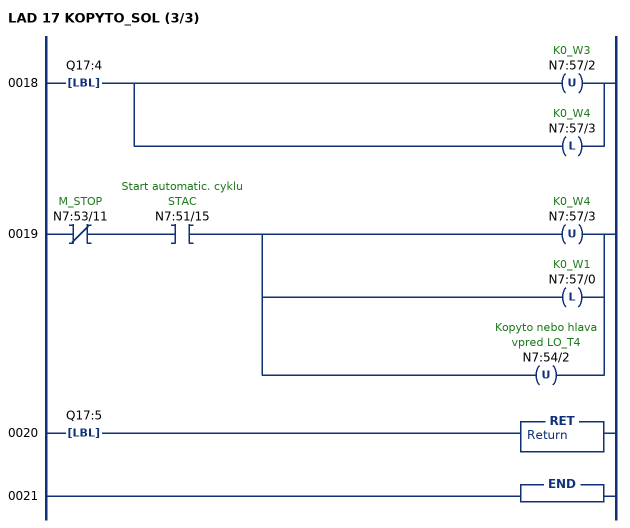
% Rung: 18 %
SOR LBL Q17:4 BST OTU N7:57/2 NXB OTL N7:57/3 BND EOR
%   N7:57/2  K0_W3 %
%   N7:57/3  K0_W4 %
% Rung: 19 %
SOR XIO N7:53/11 XIC N7:51/15 BST OTU N7:57/3 NXB OTL N7:57/0 NXB OTU N7:54/2 BND EOR
%   N7:53/11  M_STOP %
%   N7:51/15  STAC  "Start automatic. cyklu" %
%   N7:57/3  K0_W4 %
%   N7:57/0  K0_W1 %
%   N7:54/2  LO_T4  "Kopyto nebo hlava vpred" %
% Rung: 20 %
SOR LBL Q17:5 RET EOR
% Rung: 21 %
SOR END EOR

LADDER 18 "HLAVA_SOLO"
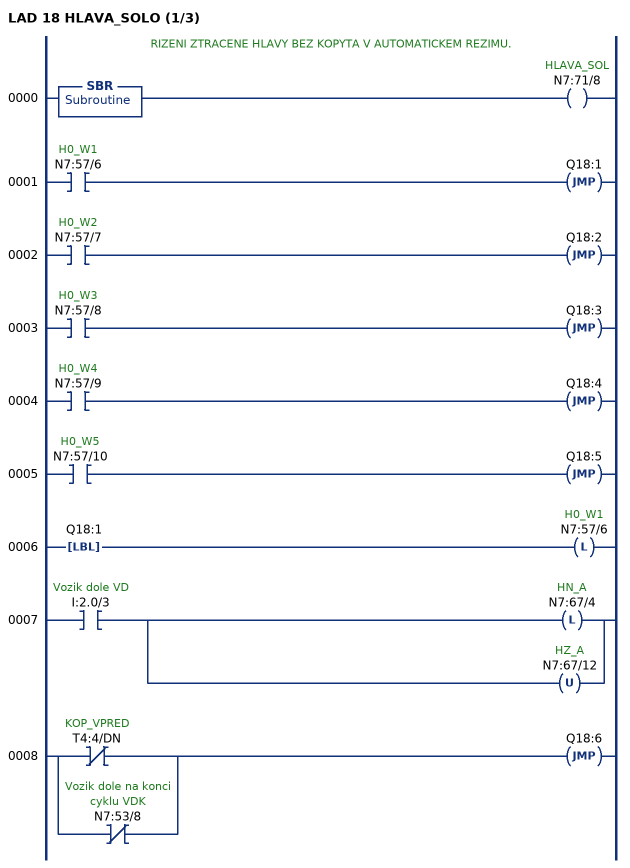
% Rung: 0 %
% RIZENI ZTRACENE HLAVY BEZ KOPYTA V AUTOMATICKEM REZIMU. %
SOR SBR OTE N7:71/8 EOR
%   N7:71/8  HLAVA_SOL %
% Rung: 1 %
SOR XIC N7:57/6 JMP Q18:1 EOR
%   N7:57/6  H0_W1 %
% Rung: 2 %
SOR XIC N7:57/7 JMP Q18:2 EOR
%   N7:57/7  H0_W2 %
% Rung: 3 %
SOR XIC N7:57/8 JMP Q18:3 EOR
%   N7:57/8  H0_W3 %
% Rung: 4 %
SOR XIC N7:57/9 JMP Q18:4 EOR
%   N7:57/9  H0_W4 %
% Rung: 5 %
SOR XIC N7:57/10 JMP Q18:5 EOR
%   N7:57/10  H0_W5 %
% Rung: 6 %
SOR LBL Q18:1 OTL N7:57/6 EOR
%   N7:57/6  H0_W1 %
% Rung: 7 %
SOR XIC I:2.0/3 BST OTL N7:67/4 NXB OTU N7:67/12 BND EOR
%   I:2.0/3  VD  "Vozik dole" %
%   N7:67/4  HN_A %
%   N7:67/12  HZ_A %
% Rung: 8 %
SOR BST XIO T4:4/DN NXB XIO N7:53/8 BND JMP Q18:6 EOR
%   T4:4/DN  KOP_VPRED %
%   N7:53/8  VDK  "Vozik dole na konci cyklu" %

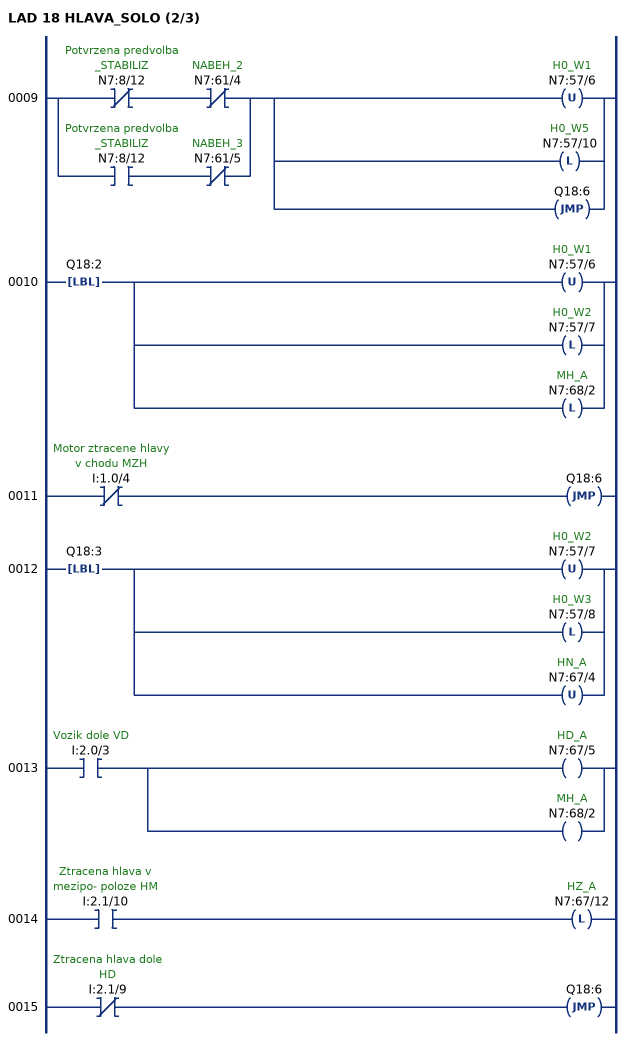
% Rung: 9 %
SOR BST XIO N7:8/12 XIO N7:61/4 NXB XIC N7:8/12 XIO N7:61/5 BND BST OTU N7:57/6 NXB BST OTL N7:57/10 NXB JMP Q18:6 BND BND EOR
%   N7:8/12  _STABILIZ  "Potvrzena predvolba" %
%   N7:61/4  NABEH_2 %
%   N7:61/5  NABEH_3 %
%   N7:57/6  H0_W1 %
%   N7:57/10  H0_W5 %
% Rung: 10 %
SOR LBL Q18:2 BST OTU N7:57/6 NXB OTL N7:57/7 NXB OTL N7:68/2 BND EOR
%   N7:57/6  H0_W1 %
%   N7:57/7  H0_W2 %
%   N7:68/2  MH_A %
% Rung: 11 %
SOR XIO I:1.0/4 JMP Q18:6 EOR
%   I:1.0/4  MZH  "Motor ztracene hlavy v chodu" %
% Rung: 12 %
SOR LBL Q18:3 BST OTU N7:57/7 NXB OTL N7:57/8 NXB OTU N7:67/4 BND EOR
%   N7:57/7  H0_W2 %
%   N7:57/8  H0_W3 %
%   N7:67/4  HN_A %
% Rung: 13 %
SOR XIC I:2.0/3 BST OTE N7:67/5 NXB OTE N7:68/2 BND EOR
%   I:2.0/3  VD  "Vozik dole" %
%   N7:67/5  HD_A %
%   N7:68/2  MH_A %
% Rung: 14 %
SOR XIC I:2.1/10 OTL N7:67/12 EOR
%   I:2.1/10  HM  "Ztracena hlava v mezipo- poloze" %
%   N7:67/12  HZ_A %
% Rung: 15 %
SOR XIO I:2.1/9 JMP Q18:6 EOR
%   I:2.1/9  HD  "Ztracena hlava dole" %

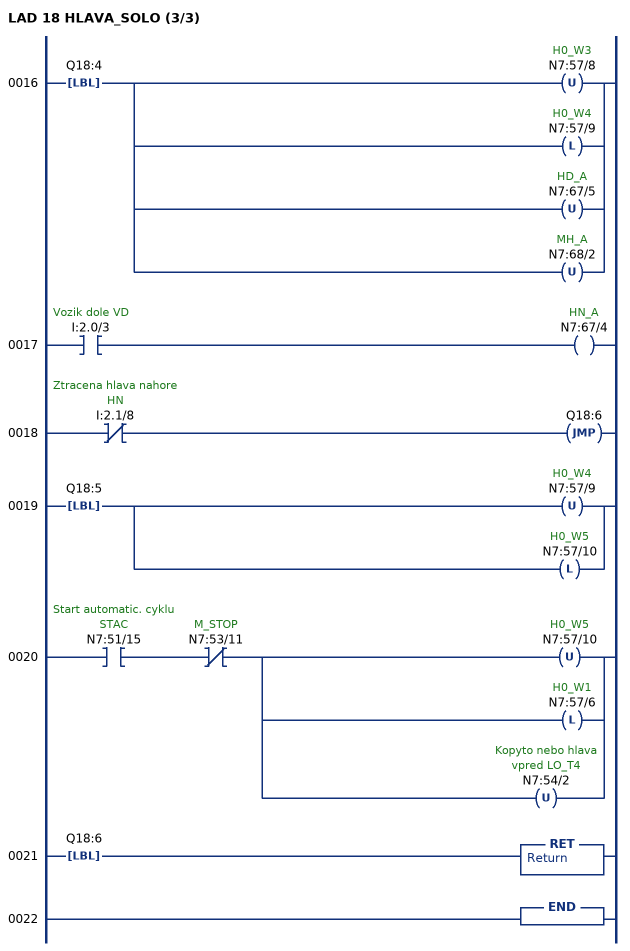
% Rung: 16 %
SOR LBL Q18:4 BST OTU N7:57/8 NXB OTL N7:57/9 NXB OTU N7:67/5 NXB OTU N7:68/2 BND EOR
%   N7:57/8  H0_W3 %
%   N7:57/9  H0_W4 %
%   N7:67/5  HD_A %
%   N7:68/2  MH_A %
% Rung: 17 %
SOR XIC I:2.0/3 OTE N7:67/4 EOR
%   I:2.0/3  VD  "Vozik dole" %
%   N7:67/4  HN_A %
% Rung: 18 %
SOR XIO I:2.1/8 JMP Q18:6 EOR
%   I:2.1/8  HN  "Ztracena hlava nahore" %
% Rung: 19 %
SOR LBL Q18:5 BST OTU N7:57/9 NXB OTL N7:57/10 BND EOR
%   N7:57/9  H0_W4 %
%   N7:57/10  H0_W5 %
% Rung: 20 %
SOR XIC N7:51/15 XIO N7:53/11 BST OTU N7:57/10 NXB OTL N7:57/6 NXB OTU N7:54/2 BND EOR
%   N7:51/15  STAC  "Start automatic. cyklu" %
%   N7:53/11  M_STOP %
%   N7:57/10  H0_W5 %
%   N7:57/6  H0_W1 %
%   N7:54/2  LO_T4  "Kopyto nebo hlava vpred" %
% Rung: 21 %
SOR LBL Q18:6 RET EOR
% Rung: 22 %
SOR END EOR

LADDER 19 "KOPY_HLAVA"
